(* PLC project Sin nombre, Desconocido Sin nombre 1 *)
(* stored: creationDateTime 2022-10-31T13:44:13, modificationDateTime 2022-11-07T20:59:54 *)

PROGRAM Lab2
  VAR
    micro AT %IW0 : INT;
    led1 AT %QX0.1 : BOOL := 0;
    led2 AT %QX0.2 : BOOL := 0;
    led3 AT %QX0.3 : BOOL := 0;
    rele AT %QX0.0 : BOOL := 0;
  END_VAR
  VAR
    TP1 : TP;
    TP2 : TP;
    TP3 : TP;
    TP4 : TP;
  END_VAR
  VAR  (* added by the conversion: wires and edge detectors of the diagram *)
    _LE14_OUT : BOOL;
  END_VAR

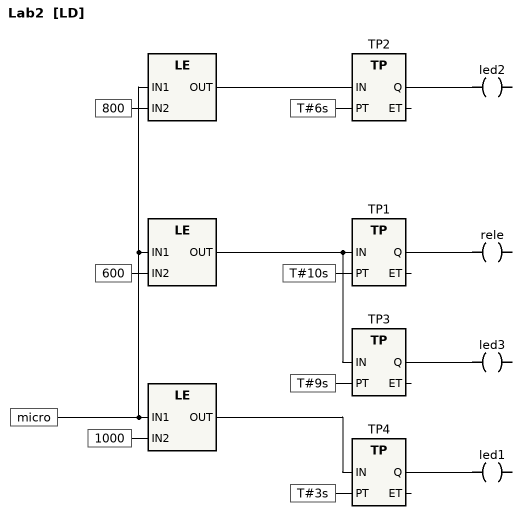
(* LD diagram, written out as Structured Text *)
_LE14_OUT := micro <= 600;
TP1(IN := _LE14_OUT, PT := T#10s);
rele := TP1.Q;
TP3(IN := _LE14_OUT, PT := T#9s);
led3 := TP3.Q;
TP2(IN := micro <= 800, PT := T#6s);
led2 := TP2.Q;
TP4(IN := micro <= 1000, PT := T#3s);
led1 := TP4.Q;
END_PROGRAM

CONFIGURATION Config0
  RESOURCE Res0 ON PLC
    TASK task0(INTERVAL := T#20ms, PRIORITY := 0);
    PROGRAM instance0 WITH task0 : Lab2;
  END_RESOURCE
END_CONFIGURATION
